// TIA Portal V18 export
FUNCTION_BLOCK "Block_1"   // FB1, LAD
{ S7_Optimized_Access := 'TRUE' }
// stored: MemoryReserve 100, SetENOAutomatically false
BEGIN

REGION Network 1
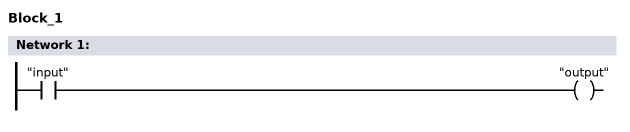
   RUNG wire#powerrail
      Contact( "input" )
      Coil( "output" )
   END_RUNG
   // the same network as SCL:
   "output" := "input";
END_REGION
END_FUNCTION_BLOCK
